FUNCTION_BLOCK PnPView (* Composite Function Block Type *)
  (* Standard: 61499-2 *)
  (* Version 0.0, 2/8/2012, XPMUser, nxtControl GmbH, template *)
  PACKAGE Main;
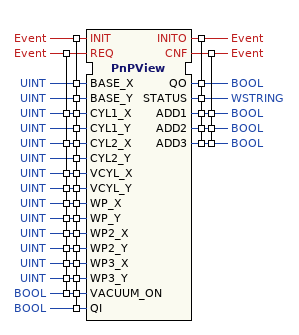
  EVENT_INPUT
    INIT WITH BASE_X, BASE_Y, CYL1_Y, CYL2_Y, CYL1_X, CYL2_X, VCYL_X, VCYL_Y, WP_X, WP_Y, VACUUM_ON, WP2_Y, WP2_X, WP3_X, WP3_Y, QI; (* Initialization Request *)
    REQ WITH CYL1_X, CYL2_X, VCYL_X, VCYL_Y, WP_X, WP_Y, VACUUM_ON, WP2_X, WP2_Y, WP3_X, WP3_Y; (* Normal Execution Request *)
  END_EVENT
  EVENT_OUTPUT
    INITO WITH QO, STATUS, ADD1, ADD2, ADD3; (* Initialization Confirm *)
    CNF WITH ADD1, ADD2, ADD3;
  END_EVENT
  VAR_INPUT
    BASE_X : UINT;
    BASE_Y : UINT;
    CYL1_X : UINT;
    CYL1_Y : UINT;
    CYL2_X : UINT;
    CYL2_Y : UINT;
    VCYL_X : UINT;
    VCYL_Y : UINT;
    WP_X : UINT;
    WP_Y : UINT;
    WP2_X : UINT;
    WP2_Y : UINT;
    WP3_X : UINT;
    WP3_Y : UINT;
    VACUUM_ON : BOOL;
    QI : BOOL;
  END_VAR
  VAR_OUTPUT
    QO : BOOL;
    STATUS : WSTRING;
    ADD1 : BOOL;
    ADD2 : BOOL;
    ADD3 : BOOL;
  END_VAR
  FBS
    IThis : PnPView_HMI;
  END_FBS
  EVENT_CONNECTIONS
    INIT TO IThis.INIT;
    REQ TO IThis.REQ;
    IThis.INITO TO INITO;
    IThis.CNF TO CNF;
    INIT TO IThis.REQ;
  END_CONNECTIONS
  DATA_CONNECTIONS
    BASE_X TO IThis.BASE_X;
    BASE_Y TO IThis.BASE_Y;
    CYL1_X TO IThis.CYL1_X;
    CYL1_Y TO IThis.CYL1_Y;
    CYL2_X TO IThis.CYL2_X;
    CYL2_Y TO IThis.CYL2_Y;
    VCYL_X TO IThis.VCYL_X;
    VCYL_Y TO IThis.VCYL_Y;
    WP_X TO IThis.WP1_X;
    WP_Y TO IThis.WP1_Y;
    WP2_X TO IThis.WP2_X;
    WP2_Y TO IThis.WP2_Y;
    WP3_X TO IThis.WP3_X;
    WP3_Y TO IThis.WP3_Y;
    VACUUM_ON TO IThis.VACUUM_ON;
    QI TO IThis.QI;
    IThis.QO TO QO;
    IThis.STATUS TO STATUS;
    IThis.ADD1 TO ADD1;
    IThis.ADD2 TO ADD2;
    IThis.ADD3 TO ADD3;
  END_CONNECTIONS
END_FUNCTION_BLOCK
